TYPE stCustomPattern :
STRUCT
	Offset_X		: ARRAY [1..24] OF INT;
	Offset_Y		: ARRAY [1..24] OF INT;
	Offset_Z		: ARRAY [1..24] OF INT;
END_STRUCT
END_TYPE

(* stored: Version 1.1.0.1, ProductVersion 3.1.4024.12
   DUT stCustomPattern: Id {12302e6b-253d-4b1c-954f-b0e2054ffad3} *)
